{attribute 'GeneratedUsingTerminal: EL3483-0060-0020'}
{attribute addProperty BoxType "EL3483-0060-0020"}
{attribute addProperty Id "EtcSlaveTerminalBaseL1_StatusAT %I*L1_Status_12B1E6BB5L1_BasicAT %I*L1_Basic_9F3F6F484L2_StatusAT %I*L2_Status_12B1E6BB5L2_BasicAT %I*L2_Basic_9F3F6F484L3_StatusAT %I*L3_Status_12B1E6BB5L3_BasicAT %I*L3_Basic_9F3F6F484Total_StatusAT %I*Total_Status_AD43C3B912Total_AdvancedAT %I*Total_Advanced_3B87F4672Total_L_L_VoltageAT %I*Total_L_L_Voltage_2881351912WcStateAT %I*WcState_9091E0EB2InfoDataAT %I*InfoData_32EB74EA10"}
{attribute addProperty CRC "593942170"}
{attribute addProperty Size "65"}
TYPE EL3483_2366D69A EXTENDS EtcSlaveTerminalBase :
STRUCT
	{attribute addProperty Name "L1_Status"}
	L1_Status : L1_Status_12B1E6BB;
	{attribute addProperty Name "L1_Basic"}
	L1_Basic : L1_Basic_9F3F6F48;
	{attribute addProperty Name "L2_Status"}
	L2_Status : L2_Status_12B1E6BB;
	{attribute addProperty Name "L2_Basic"}
	L2_Basic : L2_Basic_9F3F6F48;
	{attribute addProperty Name "L3_Status"}
	L3_Status : L3_Status_12B1E6BB;
	{attribute addProperty Name "L3_Basic"}
	L3_Basic : L3_Basic_9F3F6F48;
	{attribute addProperty Name "Total_Status"}
	Total_Status : Total_Status_AD43C3B9;
	{attribute addProperty Name "Total_Advanced"}
	Total_Advanced : Total_Advanced_3B87F467;
	{attribute addProperty Name "Total_L_L_Voltage"}
	Total_L_L_Voltage : Total_L_L_Voltage_28813519;
	{attribute addProperty Name "WcState"}
	WcState : WcState_9091E0EB;
	{attribute addProperty Name "InfoData"}
	InfoData : InfoData_32EB74EA;
END_STRUCT
END_TYPE

(* stored: Version 1.2.0.0, ProductVersion 3.1.4024.9
   DUT EL3483_2366D69A: Id {3c3dbd09-029b-490d-af04-2f46ee941f90} *)
